TYPE
    ST_RecoveryBoardList : STRUCT
        BoardID : STRING;
        Index   : STRING;
        Length  : STRING;
    END_STRUCT
END_TYPE

(* stored: Version 1.1.0.1
   DUT ST_RecoveryBoardList: Id {aa6e8fe8-9fd4-4438-8e97-0c96416e5d8c} *)
